KUKA KRL program: ps_b_ltb_res_c03.src, ps_b_ltb_res_c03.dat

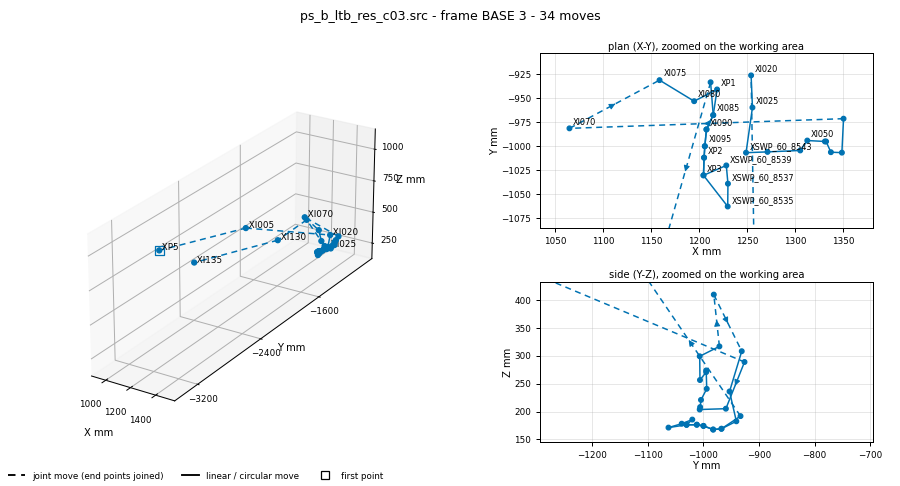
[picture p0: tool path of ps_b_ltb_res_c03.src in frame BASE 3, 34 of 34 moves have a stored position in this frame; points joined in program order, loops and branches not executed]
--- ps_b_ltb_res_c03.src ---
&ACCESS RVO1
&REL 4
&COMMENT Solda Axor LTB
&PARAM DISKPATH = KRC:\R1\Program\OLP
DEF ps_b_ltb_res_c03( )

;FOLD INI
;FOLD SPOTTECH INI
USERSPOT(#INIT)
;ENDFOLD (SPOTTECH INI)
;FOLD GRIPPERTECH INI
USER_GRP(0,DUMMY,DUMMY,GDEFAULT)
;ENDFOLD (GRIPPERTECH INI)
  ;FOLD USER INI
    ;Make your modifications here

  ;ENDFOLD (USER INI)
;ENDFOLD (INI)

; Caracterizacao dos meios de producao
; Changes: Solda Respot - AXOR - LTB
; Versao Atual: 18/02/2016
; Ferramenta: Gun C3
; Name: P13.060-R1

chk_w4_wechs_ok ( )     ; CHECK GUN C3

IF (NOT(GHOST())) THEN
IF MaxStandMenge(4) THEN
  MaxStandmengeErreicht(4)
ENDIF
IF Elektrodenwechsel(4) THEN
  e_Fraes_4 ()
ENDIF
ENDIF

;FOLD PTP P5 Vel=100 % PDAT2 Tool[4]:PINCA C3 Base[3]:Atego/Axor;%{PE}%R 8.2.20,%MKUKATPBASIS,%CMOVE,%VPTP,%P 1:PTP, 2:P5, 3:, 5:100, 7:PDAT2
$BWDSTART=FALSE
PDAT_ACT=PPDAT2
FDAT_ACT=FP5
BAS(#PTP_PARAMS,100)
PTP XP5
;ENDFOLD

;FOLD OUT 3380 'Perfil Livre Estacao' State=FALSE ;%{PE}%R 8.2.20,%MKUKATPBASIS,%COUT,%VOUTX,%P 2:3380, 3:Perfil Livre Estacao, 5:FALSE, 6:
$OUT[3380]=FALSE
;ENDFOLD

;FOLD ; Liga intertravamento 12 com R5;%{PE}%R 8.2.20,%MKUKATPBASIS,%CCOMMENT,%VNORMAL,%P 2:Liga  intertravamento  12  com  R5
;ENDFOLD
;FOLD Collision.Monitoring_12_On ;%{PE}%MKUKATPUSER
COLLSTOP( 12, 1 ) ;not Interrupt-Controlled
;ENDFOLD

;FOLD ; Liga intertravamento 13 com R5;%{PE}%R 8.2.20,%MKUKATPBASIS,%CCOMMENT,%VNORMAL,%P 2:Liga  intertravamento  13  com  R5
;ENDFOLD
;FOLD Collision.Monitoring_13_On ;%{PE}%MKUKATPUSER
COLLSTOP( 13, 1 ) ;not Interrupt-Controlled
;ENDFOLD

;FOLD PTP l005 CONT Vel=100 % P_OLP2 Tool[4]:PINCA C3 Base[3]:Atego/Axor;%{PE}%R 8.2.20,%MKUKATPBASIS,%CMOVE,%VPTP,%P 1:PTP, 2:l005, 3:C_DIS, 5:100, 7:P_OLP2
$BWDSTART=FALSE
PDAT_ACT=PP_OLP2
FDAT_ACT=Fl005
BAS(#PTP_PARAMS,100)
PTP Xl005 C_DIS
;ENDFOLD
;FOLD PTP l020 CONT Vel=100 % PDAT3 Tool[4]:PINCA C3 Base[3]:Atego/Axor;%{PE}%R 8.2.20,%MKUKATPBASIS,%CMOVE,%VPTP,%P 1:PTP, 2:l020, 3:C_DIS, 5:100, 7:PDAT3
$BWDSTART=FALSE
PDAT_ACT=PPDAT3
FDAT_ACT=Fl020
BAS(#PTP_PARAMS,100)
PTP Xl020 C_DIS
;ENDFOLD
;FOLD LIN l025 CONT Vel=2 m/s L_OLP3 Tool[4]:PINCA C3 Base[3]:Atego/Axor;%{PE}%R 8.2.20,%MKUKATPBASIS,%CMOVE,%VLIN,%P 1:LIN, 2:l025, 3:C_DIS C_DIS, 5:2, 7:L_OLP3
$BWDSTART=FALSE
LDAT_ACT=LL_OLP3
FDAT_ACT=Fl025
BAS(#CP_PARAMS,2)
LIN Xl025 C_DIS C_DIS
;ENDFOLD

;FOLD ; SWP_60_8543;%{PE}%R 4.1.16,%MKUKATPBASIS,%CCOMMENT,%VNORMAL,%P 2:SWP_60_8543
;ENDFOLD
;FOLD LIN SWP_60_8543 L_OLP4 SPOT Gun=3 RETR CLS PgNo1=196 ACTIVE=1 Tool[4]:PINCA C3 Base[3]:Atego/Axor;%{PE}%R 8.2.2,%MKUKATPSPOT,%CSPOT,%VLIN,%P 1:LIN, 2:SWP_60_8543, 3:, 5:2, 7:L_OLP4, 10:3, 12:#FIRST, 14:#CLO, 16:196, 18:1, 20:0, 22:0, 24:1, 25:NORMAL
$BWDSTART=FALSE
LDAT_ACT=LL_OLP4
FDAT_ACT=FSWP_60_8543
BAS(#CP_PARAMS,LL_OLP4.VEL)
S_ACT.GUN=3
S_ACT.PAIR=SDEFAULT.PAIR
S_ACT.RETR=#CLO
S_ACT.CLO_TM=1
S_ACT.PGNO1=196
S_ACT.PGNO2=SDEFAULT.PGNO2
S_ACT.PRESS1=SDEFAULT.PRESS1
S_ACT.PRESS2=SDEFAULT.PRESS2
S_READY=FALSE
LIN XSWP_60_8543
USERSPOT(#SPOT, S_ACT)
WAIT FOR S_READY
;ENDFOLD

;FOLD ; SWP_60_8545;%{PE}%R 4.1.16,%MKUKATPBASIS,%CCOMMENT,%VNORMAL,%P 2:SWP_60_8545
;ENDFOLD
;FOLD LIN SWP_60_8545 L_OLP8 SPOT Gun=3 RETR CLS PgNo1=196 ACTIVE=1 Tool[4]:PINCA C3 Base[3]:Atego/Axor;%{PE}%R 8.2.2,%MKUKATPSPOT,%CSPOT,%VLIN,%P 1:LIN, 2:SWP_60_8545, 3:, 5:2, 7:L_OLP8, 10:3, 12:#FIRST, 14:#CLO, 16:196, 18:1, 20:0, 22:0, 24:1, 25:NORMAL
$BWDSTART=FALSE
LDAT_ACT=LL_OLP8
FDAT_ACT=FSWP_60_8545
BAS(#CP_PARAMS,LL_OLP8.VEL)
S_ACT.GUN=3
S_ACT.PAIR=SDEFAULT.PAIR
S_ACT.RETR=#CLO
S_ACT.CLO_TM=1
S_ACT.PGNO1=196
S_ACT.PGNO2=SDEFAULT.PGNO2
S_ACT.PRESS1=SDEFAULT.PRESS1
S_ACT.PRESS2=SDEFAULT.PRESS2
S_READY=FALSE
LIN XSWP_60_8545
USERSPOT(#SPOT, S_ACT)
WAIT FOR S_READY
;ENDFOLD

;FOLD ; SWP_60_8547;%{PE}%R 4.1.16,%MKUKATPBASIS,%CCOMMENT,%VNORMAL,%P 2:SWP_60_8547
;ENDFOLD
;FOLD LIN SWP_60_8547 L_OLP9 SPOT Gun=3 RETR CLS PgNo1=196 ACTIVE=1 Tool[4]:PINCA C3 Base[3]:Atego/Axor;%{PE}%R 8.2.2,%MKUKATPSPOT,%CSPOT,%VLIN,%P 1:LIN, 2:SWP_60_8547, 3:, 5:2, 7:L_OLP9, 10:3, 12:#FIRST, 14:#CLO, 16:196, 18:1, 20:0, 22:0, 24:1, 25:NORMAL
$BWDSTART=FALSE
LDAT_ACT=LL_OLP9
FDAT_ACT=FSWP_60_8547
BAS(#CP_PARAMS,LL_OLP9.VEL)
S_ACT.GUN=3
S_ACT.PAIR=SDEFAULT.PAIR
S_ACT.RETR=#CLO
S_ACT.CLO_TM=1
S_ACT.PGNO1=196
S_ACT.PGNO2=SDEFAULT.PGNO2
S_ACT.PRESS1=SDEFAULT.PRESS1
S_ACT.PRESS2=SDEFAULT.PRESS2
S_READY=FALSE
LIN XSWP_60_8547
USERSPOT(#SPOT, S_ACT)
WAIT FOR S_READY
;ENDFOLD

;FOLD LIN l050 CONT Vel=2 m/s L_OLP10 Tool[4]:PINCA C3 Base[3]:Atego/Axor;%{PE}%R 8.2.20,%MKUKATPBASIS,%CMOVE,%VLIN,%P 1:LIN, 2:l050, 3:C_DIS C_DIS, 5:2, 7:L_OLP10
$BWDSTART=FALSE
LDAT_ACT=LL_OLP10
FDAT_ACT=Fl050
BAS(#CP_PARAMS,2)
LIN Xl050 C_DIS C_DIS
;ENDFOLD
;FOLD LIN l055 CONT Vel=2 m/s L_OLP11 Tool[4]:PINCA C3 Base[3]:Atego/Axor;%{PE}%R 8.2.20,%MKUKATPBASIS,%CMOVE,%VLIN,%P 1:LIN, 2:l055, 3:C_DIS C_DIS, 5:2, 7:L_OLP11
$BWDSTART=FALSE
LDAT_ACT=LL_OLP11
FDAT_ACT=Fl055
BAS(#CP_PARAMS,2)
LIN Xl055 C_DIS C_DIS
;ENDFOLD
;FOLD LIN l025S CONT Vel=2 m/s L_OLP12 Tool[4]:PINCA C3 Base[3]:Atego/Axor;%{PE}%R 8.2.20,%MKUKATPBASIS,%CMOVE,%VLIN,%P 1:LIN, 2:l025S, 3:C_DIS C_DIS, 5:2, 7:L_OLP12
$BWDSTART=FALSE
LDAT_ACT=LL_OLP12
FDAT_ACT=Fl025S
BAS(#CP_PARAMS,2)
LIN Xl025S C_DIS C_DIS
;ENDFOLD

;FOLD ; SWP_60_8549;%{PE}%R 4.1.16,%MKUKATPBASIS,%CCOMMENT,%VNORMAL,%P 2:SWP_60_8549
;ENDFOLD
;FOLD LIN SWP_60_8549 L_OLP13 SPOT Gun=3 RETR CLS PgNo1=196 ACTIVE=1 Tool[4]:PINCA C3 Base[3]:Atego/Axor;%{PE}%R 8.2.2,%MKUKATPSPOT,%CSPOT,%VLIN,%P 1:LIN, 2:SWP_60_8549, 3:, 5:2, 7:L_OLP13, 10:3, 12:#FIRST, 14:#CLO, 16:196, 18:1, 20:0, 22:0, 24:1, 25:NORMAL
$BWDSTART=FALSE
LDAT_ACT=LL_OLP13
FDAT_ACT=FSWP_60_8549
BAS(#CP_PARAMS,LL_OLP13.VEL)
S_ACT.GUN=3
S_ACT.PAIR=SDEFAULT.PAIR
S_ACT.RETR=#CLO
S_ACT.CLO_TM=1
S_ACT.PGNO1=196
S_ACT.PGNO2=SDEFAULT.PGNO2
S_ACT.PRESS1=SDEFAULT.PRESS1
S_ACT.PRESS2=SDEFAULT.PRESS2
S_READY=FALSE
LIN XSWP_60_8549
USERSPOT(#SPOT, S_ACT)
WAIT FOR S_READY
;ENDFOLD

;FOLD ; SWP_60_8551;%{PE}%R 4.1.16,%MKUKATPBASIS,%CCOMMENT,%VNORMAL,%P 2:SWP_60_8551
;ENDFOLD
;FOLD LIN SWP_60_8551 L_OLP14 SPOT Gun=3 RETR OPN PgNo1=196 ACTIVE=1 Tool[4]:PINCA C3 Base[3]:Atego/Axor;%{PE}%R 8.2.2,%MKUKATPSPOT,%CSPOT,%VLIN,%P 1:LIN, 2:SWP_60_8551, 3:, 5:2, 7:L_OLP14, 10:3, 12:#FIRST, 14:#OPN, 16:196, 18:1, 20:0, 22:0, 24:1, 25:NORMAL
$BWDSTART=FALSE
LDAT_ACT=LL_OLP14
FDAT_ACT=FSWP_60_8551
BAS(#CP_PARAMS,LL_OLP14.VEL)
S_ACT.GUN=3
S_ACT.PAIR=SDEFAULT.PAIR
S_ACT.RETR=#OPN
S_ACT.CLO_TM=1
S_ACT.PGNO1=196
S_ACT.PGNO2=SDEFAULT.PGNO2
S_ACT.PRESS1=SDEFAULT.PRESS1
S_ACT.PRESS2=SDEFAULT.PRESS2
S_READY=FALSE
LIN XSWP_60_8551
USERSPOT(#SPOT, S_ACT)
WAIT FOR S_READY
;ENDFOLD

;FOLD LIN l065 CONT Vel=2 m/s L_OLP15 Tool[4]:PINCA C3 Base[3]:Atego/Axor;%{PE}%R 8.2.20,%MKUKATPBASIS,%CMOVE,%VLIN,%P 1:LIN, 2:l065, 3:C_DIS C_DIS, 5:2, 7:L_OLP15
$BWDSTART=FALSE
LDAT_ACT=LL_OLP15
FDAT_ACT=Fl065
BAS(#CP_PARAMS,2)
LIN Xl065 C_DIS C_DIS
;ENDFOLD
;FOLD PTP l070 CONT Vel=100 % P_OLP5 Tool[4]:PINCA C3 Base[3]:Atego/Axor;%{PE}%R 8.2.20,%MKUKATPBASIS,%CMOVE,%VPTP,%P 1:PTP, 2:l070, 3:C_DIS, 5:100, 7:P_OLP5
$BWDSTART=FALSE
PDAT_ACT=PP_OLP5
FDAT_ACT=Fl070
BAS(#PTP_PARAMS,100)
PTP Xl070 C_DIS
;ENDFOLD
;FOLD PTP l075 CONT Vel=100 % P_OLP6 Tool[4]:PINCA C3 Base[3]:Atego/Axor;%{PE}%R 8.2.20,%MKUKATPBASIS,%CMOVE,%VPTP,%P 1:PTP, 2:l075, 3:C_DIS, 5:100, 7:P_OLP6
$BWDSTART=FALSE
PDAT_ACT=PP_OLP6
FDAT_ACT=Fl075
BAS(#PTP_PARAMS,100)
PTP Xl075 C_DIS
;ENDFOLD
;FOLD LIN l080 CONT Vel=2 m/s L_OLP16 Tool[4]:PINCA C3 Base[3]:Atego/Axor;%{PE}%R 8.2.20,%MKUKATPBASIS,%CMOVE,%VLIN,%P 1:LIN, 2:l080, 3:C_DIS C_DIS, 5:2, 7:L_OLP16
$BWDSTART=FALSE
LDAT_ACT=LL_OLP16
FDAT_ACT=Fl080
BAS(#CP_PARAMS,2)
LIN Xl080 C_DIS C_DIS
;ENDFOLD
;FOLD LIN P1 CONT Vel=2 m/s CPDAT1 Tool[4]:PINCA C3 Base[3]:Atego/Axor;%{PE}%R 8.2.20,%MKUKATPBASIS,%CMOVE,%VLIN,%P 1:LIN, 2:P1, 3:C_DIS C_DIS, 5:2, 7:CPDAT1
$BWDSTART=FALSE
LDAT_ACT=LCPDAT1
FDAT_ACT=FP1
BAS(#CP_PARAMS,2)
LIN XP1 C_DIS C_DIS
;ENDFOLD
;FOLD LIN l085 Vel=2 m/s L_OLP17 Tool[4]:PINCA C3 Base[3]:Atego/Axor;%{PE}%R 8.2.20,%MKUKATPBASIS,%CMOVE,%VLIN,%P 1:LIN, 2:l085, 3:, 5:2, 7:L_OLP17
$BWDSTART=FALSE
LDAT_ACT=LL_OLP17
FDAT_ACT=Fl085
BAS(#CP_PARAMS,2)
LIN Xl085
;ENDFOLD
;FOLD LIN l090 CONT Vel=2 m/s L_OLP18 Tool[4]:PINCA C3 Base[3]:Atego/Axor;%{PE}%R 8.2.20,%MKUKATPBASIS,%CMOVE,%VLIN,%P 1:LIN, 2:l090, 3:C_DIS C_DIS, 5:2, 7:L_OLP18
$BWDSTART=FALSE
LDAT_ACT=LL_OLP18
FDAT_ACT=Fl090
BAS(#CP_PARAMS,2)
LIN Xl090 C_DIS C_DIS
;ENDFOLD
;FOLD LIN l095 CONT Vel=2 m/s L_OLP19 Tool[4]:PINCA C3 Base[3]:Atego/Axor;%{PE}%R 8.2.20,%MKUKATPBASIS,%CMOVE,%VLIN,%P 1:LIN, 2:l095, 3:C_DIS C_DIS, 5:2, 7:L_OLP19
$BWDSTART=FALSE
LDAT_ACT=LL_OLP19
FDAT_ACT=Fl095
BAS(#CP_PARAMS,2)
LIN Xl095 C_DIS C_DIS
;ENDFOLD
;FOLD LIN P2 CONT Vel=2 m/s CPDAT2 Tool[4]:PINCA C3 Base[3]:Atego/Axor;%{PE}%R 8.2.20,%MKUKATPBASIS,%CMOVE,%VLIN,%P 1:LIN, 2:P2, 3:C_DIS C_DIS, 5:2, 7:CPDAT2
$BWDSTART=FALSE
LDAT_ACT=LCPDAT2
FDAT_ACT=FP2
BAS(#CP_PARAMS,2)
LIN XP2 C_DIS C_DIS
;ENDFOLD
;FOLD LIN P3 CONT Vel=2 m/s CPDAT3 Tool[4]:PINCA C3 Base[3]:Atego/Axor;%{PE}%R 8.2.20,%MKUKATPBASIS,%CMOVE,%VLIN,%P 1:LIN, 2:P3, 3:C_DIS C_DIS, 5:2, 7:CPDAT3
$BWDSTART=FALSE
LDAT_ACT=LCPDAT3
FDAT_ACT=FP3
BAS(#CP_PARAMS,2)
LIN XP3 C_DIS C_DIS
;ENDFOLD

;FOLD ; SWP_60_8535;%{PE}%R 8.2.20,%MKUKATPBASIS,%CCOMMENT,%VNORMAL,%P 2:SWP_60_8535
;ENDFOLD
;FOLD LIN SWP_60_8535 L_OLP30 SPOT Gun=3 RETR CLS PgNo1=197 ACTIVE=1 Tool[4]:PINCA C3 Base[3]:Atego/Axor;%{PE}%R 8.2.2,%MKUKATPSPOT,%CSPOT,%VLIN,%P 1:LIN, 2:SWP_60_8535, 3:, 5:2, 7:L_OLP30, 10:3, 12:#FIRST, 14:#CLO, 16:197, 18:1, 20:0, 22:0, 24:1, 25:NORMAL
$BWDSTART=FALSE
LDAT_ACT=LL_OLP30
FDAT_ACT=FSWP_60_8535
BAS(#CP_PARAMS,LL_OLP30.VEL)
S_ACT.GUN=3
S_ACT.PAIR=SDEFAULT.PAIR
S_ACT.RETR=#CLO
S_ACT.CLO_TM=1
S_ACT.PGNO1=197
S_ACT.PGNO2=SDEFAULT.PGNO2
S_ACT.PRESS1=SDEFAULT.PRESS1
S_ACT.PRESS2=SDEFAULT.PRESS2
S_READY=FALSE
LIN XSWP_60_8535
USERSPOT(#SPOT, S_ACT)
WAIT FOR S_READY
;ENDFOLD

;FOLD ; SWP_60_8537;%{PE}%R 8.2.20,%MKUKATPBASIS,%CCOMMENT,%VNORMAL,%P 2:SWP_60_8537
;ENDFOLD
;FOLD LIN SWP_60_8537 L_OLP31 SPOT Gun=3 RETR CLS PgNo1=197 ACTIVE=1 Tool[4]:PINCA C3 Base[3]:Atego/Axor;%{PE}%R 8.2.2,%MKUKATPSPOT,%CSPOT,%VLIN,%P 1:LIN, 2:SWP_60_8537, 3:, 5:2, 7:L_OLP31, 10:3, 12:#FIRST, 14:#CLO, 16:197, 18:1, 20:0, 22:0, 24:1, 25:NORMAL
$BWDSTART=FALSE
LDAT_ACT=LL_OLP31
FDAT_ACT=FSWP_60_8537
BAS(#CP_PARAMS,LL_OLP31.VEL)
S_ACT.GUN=3
S_ACT.PAIR=SDEFAULT.PAIR
S_ACT.RETR=#CLO
S_ACT.CLO_TM=1
S_ACT.PGNO1=197
S_ACT.PGNO2=SDEFAULT.PGNO2
S_ACT.PRESS1=SDEFAULT.PRESS1
S_ACT.PRESS2=SDEFAULT.PRESS2
S_READY=FALSE
LIN XSWP_60_8537
USERSPOT(#SPOT, S_ACT)
WAIT FOR S_READY
;ENDFOLD

;FOLD ; SWP_60_8539;%{PE}%R 4.1.16,%MKUKATPBASIS,%CCOMMENT,%VNORMAL,%P 2:SWP_60_8539
;ENDFOLD
;FOLD LIN SWP_60_8539 L_OLP20 SPOT Gun=3 RETR OPN PgNo1=197 ACTIVE=1 Tool[4]:PINCA C3 Base[3]:Atego/Axor;%{PE}%R 8.2.2,%MKUKATPSPOT,%CSPOT,%VLIN,%P 1:LIN, 2:SWP_60_8539, 3:, 5:2, 7:L_OLP20, 10:3, 12:#FIRST, 14:#OPN, 16:197, 18:1, 20:0, 22:0, 24:1, 25:NORMAL
$BWDSTART=FALSE
LDAT_ACT=LL_OLP20
FDAT_ACT=FSWP_60_8539
BAS(#CP_PARAMS,LL_OLP20.VEL)
S_ACT.GUN=3
S_ACT.PAIR=SDEFAULT.PAIR
S_ACT.RETR=#OPN
S_ACT.CLO_TM=1
S_ACT.PGNO1=197
S_ACT.PGNO2=SDEFAULT.PGNO2
S_ACT.PRESS1=SDEFAULT.PRESS1
S_ACT.PRESS2=SDEFAULT.PRESS2
S_READY=FALSE
LIN XSWP_60_8539
USERSPOT(#SPOT, S_ACT)
WAIT FOR S_READY
;ENDFOLD

;FOLD LIN P4 CONT Vel=2 m/s CPDAT4 Tool[4]:PINCA C3 Base[3]:Atego/Axor;%{PE}%R 8.2.20,%MKUKATPBASIS,%CMOVE,%VLIN,%P 1:LIN, 2:P4, 3:C_DIS C_DIS, 5:2, 7:CPDAT4
$BWDSTART=FALSE
LDAT_ACT=LCPDAT4
FDAT_ACT=FP4
BAS(#CP_PARAMS,2)
LIN XP4 C_DIS C_DIS
;ENDFOLD
;FOLD LIN l100 CONT Vel=2 m/s L_OLP23 Tool[4]:PINCA C3 Base[3]:Atego/Axor;%{PE}%R 8.2.20,%MKUKATPBASIS,%CMOVE,%VLIN,%P 1:LIN, 2:l100, 3:C_DIS C_DIS, 5:2, 7:L_OLP23
$BWDSTART=FALSE
LDAT_ACT=LL_OLP23
FDAT_ACT=Fl100
BAS(#CP_PARAMS,2)
LIN Xl100 C_DIS C_DIS
;ENDFOLD
;FOLD LIN l105 CONT Vel=2 m/s L_OLP24 Tool[4]:PINCA C3 Base[3]:Atego/Axor;%{PE}%R 8.2.20,%MKUKATPBASIS,%CMOVE,%VLIN,%P 1:LIN, 2:l105, 3:C_DIS C_DIS, 5:2, 7:L_OLP24
$BWDSTART=FALSE
LDAT_ACT=LL_OLP24
FDAT_ACT=Fl105
BAS(#CP_PARAMS,2)
LIN Xl105 C_DIS C_DIS
;ENDFOLD
;FOLD LIN l110 CONT Vel=2 m/s L_OLP25 Tool[4]:PINCA C3 Base[3]:Atego/Axor;%{PE}%R 8.2.20,%MKUKATPBASIS,%CMOVE,%VLIN,%P 1:LIN, 2:l110, 3:C_DIS C_DIS, 5:2, 7:L_OLP25
$BWDSTART=FALSE
LDAT_ACT=LL_OLP25
FDAT_ACT=Fl110
BAS(#CP_PARAMS,2)
LIN Xl110 C_DIS C_DIS
;ENDFOLD
;FOLD LIN l115  Vel=2.00 m/s L_OLP26 Tool[4]:Gun C03 Base[3]:Atego/Axor;%{PE}%R8.2.19,%MKUKATPBASIS,%CMOVE,%VLIN,%P 1:LIN, 2:l115, 3: , 5:2.00, 7:L_OLP26
$BWDSTART = FALSE
LDAT_ACT= LL_OLP26
FDAT_ACT= Fl115
BAS(#CP_PARAMS,2.00)
LIN Xl115
;ENDFOLD
;FOLD LIN l120 CONT Vel=2 m/s L_OLP27 Tool[4]:PINCA C3 Base[3]:Atego/Axor;%{PE}%R 8.2.20,%MKUKATPBASIS,%CMOVE,%VLIN,%P 1:LIN, 2:l120, 3:C_DIS C_DIS, 5:2, 7:L_OLP27
$BWDSTART=FALSE
LDAT_ACT=LL_OLP27
FDAT_ACT=Fl120
BAS(#CP_PARAMS,2)
LIN Xl120 C_DIS C_DIS
;ENDFOLD
;FOLD PTP l125 CONT Vel=100 % PDAT4 Tool[4]:PINCA C3 Base[3]:Atego/Axor;%{PE}%R 8.2.20,%MKUKATPBASIS,%CMOVE,%VPTP,%P 1:PTP, 2:l125, 3:C_DIS, 5:100, 7:PDAT4
$BWDSTART=FALSE
PDAT_ACT=PPDAT4
FDAT_ACT=Fl125
BAS(#PTP_PARAMS,100)
PTP Xl125 C_DIS
;ENDFOLD
;FOLD PTP l130 CONT Vel=100 % PDAT5 Tool[4]:PINCA C3 Base[3]:Atego/Axor;%{PE}%R 8.2.20,%MKUKATPBASIS,%CMOVE,%VPTP,%P 1:PTP, 2:l130, 3:C_DIS, 5:100, 7:PDAT5
$BWDSTART=FALSE
PDAT_ACT=PPDAT5
FDAT_ACT=Fl130
BAS(#PTP_PARAMS,100)
PTP Xl130 C_DIS
;ENDFOLD
;FOLD PTP l135 Vel=100 % P_OLP7 Tool[4]:PINCA C3 Base[3]:Atego/Axor;%{PE}%R 8.2.20,%MKUKATPBASIS,%CMOVE,%VPTP,%P 1:PTP, 2:l135, 3:, 5:100, 7:P_OLP7
$BWDSTART=FALSE
PDAT_ACT=PP_OLP7
FDAT_ACT=Fl135
BAS(#PTP_PARAMS,100)
PTP Xl135
;ENDFOLD

;FOLD ; Desliga intertravamento 12 com R5;%{PE}%R 8.2.20,%MKUKATPBASIS,%CCOMMENT,%VNORMAL,%P 2:Desliga  intertravamento  12  com  R5
;ENDFOLD
;FOLD Collision.Monitoring_12_Off . ;%{PE}%MKUKATPUSER
COLLSTOP( 12, 2+0 )
;ENDFOLD

;FOLD ; Desliga intertravamento 13 com R5;%{PE}%R 8.2.20,%MKUKATPBASIS,%CCOMMENT,%VNORMAL,%P 2:Desliga  intertravamento  13  com  R5
;ENDFOLD
;FOLD Collision.Monitoring_13_Off . ;%{PE}%MKUKATPUSER
COLLSTOP( 13, 2+0 )
;ENDFOLD

end_weld_respot ()

IF (NOT(GHOST())) THEN
IF FraesAnf(4) THEN
  f_Fraes_4 ()
ENDIF
ENDIF

END

--- ps_b_ltb_res_c03.dat ---
&ACCESS RVO1
&REL 4
&COMMENT Solda Axor LTB
&PARAM DISKPATH = KRC:\R1\Program\OLP
DEFDAT ps_b_ltb_res_c03
;FOLD EXTERNAL DECLARATIONS;%{PE}%MKUKATPBASIS,%CEXT,%VCOMMON,%P
;FOLD GRIPPERTECH EXT
EXT  H50 (INT  :IN,INT  :IN,INT  :IN,GRP_TYP  :IN )
;ENDFOLD (GRIPPERTECH EXT)
;FOLD SPOTTECH EXT
EXT  USERSPOT (S_COMMAND  :IN,SPOT_TYPE  :IN )
;ENDFOLD (SPOTTECH EXT)
;FOLD BASISTECH EXT;%{PE}%MKUKATPBASIS,%CEXT,%VEXT,%P
EXT  BAS (BAS_COMMAND  :IN,REAL  :IN )
DECL INT SUCCESS
;ENDFOLD (BASISTECH EXT)
;FOLD USER EXT;%{E}%MKUKATPUSER,%CEXT,%VEXT,%P
;Make your modifications here

;ENDFOLD (USER EXT)
;ENDFOLD (EXTERNAL DECLARATIONS)
DECL FDAT Fl005={TOOL_NO 4,BASE_NO 3,IPO_FRAME #BASE,POINT2[] " "}
DECL PDAT PP_OLP2={VEL 100.0,ACC 100.0,APO_DIST 200.0,APO_MODE #CDIS}
DECL E6POS Xl005={X 1274.78198,Y -2152.4519,Z 802.703003,A 0.067400001,B 28.0000992,C 90.0,S 2,T 11}
DECL FDAT Fl020={TOOL_NO 4,BASE_NO 3,IPO_FRAME #BASE,POINT2[] " "}
DECL E6POS Xl020={X 1253.90295,Y -926.031982,Z 289.157806,A 0.0670686066,B 27.9958591,C 89.9981689,S 18,T 11,E1 0.0,E2 0.0,E3 0.0,E4 0.0,E5 0.0,E6 0.0}
DECL FDAT Fl025={TOOL_NO 4,BASE_NO 3,IPO_FRAME #BASE,POINT2[] " "}
DECL E6POS Xl025={X 1255.30298,Y -959.498718,Z 205.282593,A 0.0679476634,B 27.99827,C 89.999649,S 18,T 11,E1 0.0,E2 0.0,E3 0.0,E4 0.0,E5 0.0,E6 0.0}
DECL LDAT LL_OLP3={VEL 2.0,ACC 100.0,APO_DIST 10.0,APO_FAC 0.0,ORI_TYP #VAR,CIRC_TYP #BASE,JERK_FAC 50.0}
DECL FDAT FSWP_60_8543={TOOL_NO 4,BASE_NO 3,IPO_FRAME #BASE,POINT2[] " "}
DECL E6POS XSWP_60_8543={X 1248.61499,Y -1006.54199,Z 203.796402,A -0.129490495,B 27.9995594,C 92.4205933,S 18,T 11,E1 0.0,E2 0.0,E3 0.0,E4 0.0,E5 0.0,E6 0.0}
DECL LDAT LL_OLP4={VEL 2.0,ACC 100.0,APO_DIST 0.0,APO_FAC 0.0,ORI_TYP #VAR,CIRC_TYP #BASE,JERK_FAC 50.0}
DECL FDAT FSWP_60_8545={TOOL_NO 4,BASE_NO 3,IPO_FRAME #BASE,POINT2[] " "}
DECL E6POS XSWP_60_8545={X 1270.98096,Y -1005.711,Z 208.158401,A -0.129547194,B 27.9999104,C 92.419487,S 18,T 11,E1 0.0,E2 0.0,E3 0.0,E4 0.0,E5 0.0,E6 0.0}
DECL LDAT LL_OLP8={VEL 2.0,ACC 100.0,APO_DIST 0.0,APO_FAC 0.0,ORI_TYP #VAR,CIRC_TYP #BASE,JERK_FAC 50.0}
DECL FDAT FSWP_60_8547={TOOL_NO 4,BASE_NO 3,IPO_FRAME #BASE,POINT2[] " "}
DECL E6POS XSWP_60_8547={X 1305.07202,Y -1004.21399,Z 221.033096,A 0.224301994,B 35.0479698,C 92.027832,S 18,T 11,E1 0.0,E2 0.0,E3 0.0,E4 0.0,E5 0.0,E6 0.0}
DECL LDAT LL_OLP9={VEL 2.0,ACC 100.0,APO_DIST 0.0,APO_FAC 0.0,ORI_TYP #VAR,CIRC_TYP #BASE,JERK_FAC 50.0}
DECL FDAT Fl050={TOOL_NO 4,BASE_NO 3,IPO_FRAME #BASE,POINT2[] " "}
DECL E6POS Xl050={X 1312.42297,Y -993.888977,Z 240.986099,A 0.0672914535,B 27.9993992,C 90.0008469,S 18,T 11,E1 0.0,E2 0.0,E3 0.0,E4 0.0,E5 0.0,E6 0.0}
DECL LDAT LL_OLP10={VEL 2.0,ACC 100.0,APO_DIST 5.0,APO_FAC 0.0,ORI_TYP #VAR,CIRC_TYP #BASE,JERK_FAC 50.0}
DECL FDAT Fl055={TOOL_NO 4,BASE_NO 3,IPO_FRAME #BASE,POINT2[] " "}
DECL E6POS Xl055={X 1330.77405,Y -994.846619,Z 273.997803,A 0.0951634571,B 19.9996204,C 90.0010986,S 18,T 11,E1 0.0,E2 0.0,E3 0.0,E4 0.0,E5 0.0,E6 0.0}
DECL LDAT LL_OLP11={VEL 2.0,ACC 100.0,APO_DIST 5.0,APO_FAC 0.0,ORI_TYP #VAR,CIRC_TYP #BASE,JERK_FAC 50.0}
DECL FDAT Fl025S={TOOL_NO 4,BASE_NO 3,IPO_FRAME #BASE,POINT2[] " "}
DECL E6POS Xl025S={X 1331.99402,Y -994.88147,Z 271.029297,A 0.0962694436,B -0.00231891288,C 89.9995804,S 18,T 11,E1 0.0,E2 0.0,E3 0.0,E4 0.0,E5 0.0,E6 0.0}
DECL LDAT LL_OLP12={VEL 2.0,ACC 100.0,APO_DIST 5.0,APO_FAC 0.0,ORI_TYP #VAR,CIRC_TYP #BASE,JERK_FAC 50.0}
DECL FDAT FSWP_60_8549={TOOL_NO 4,BASE_NO 3,IPO_FRAME #BASE,POINT2[] " "}
DECL E6POS XSWP_60_8549={X 1336.99695,Y -1006.02899,Z 256.759003,A 2.13942194,B -0.046111729,C 91.2335129,S 18,T 3,E1 0.0,E2 0.0,E3 0.0,E4 0.0,E5 0.0,E6 0.0}
DECL LDAT LL_OLP13={VEL 2.0,ACC 100.0,APO_DIST 0.0,APO_FAC 0.0,ORI_TYP #VAR,CIRC_TYP #BASE,JERK_FAC 50.0}
DECL FDAT FSWP_60_8551={TOOL_NO 4,BASE_NO 3,IPO_FRAME #BASE,POINT2[] " "}
DECL E6POS XSWP_60_8551={X 1348.448,Y -1006.50098,Z 299.4151,A 0.931857288,B -0.001559027,C 90.0008163,S 18,T 11,E1 0.0,E2 0.0,E3 0.0,E4 0.0,E5 0.0,E6 0.0}
DECL LDAT LL_OLP14={VEL 2.0,ACC 100.0,APO_DIST 0.0,APO_FAC 0.0,ORI_TYP #VAR,CIRC_TYP #BASE,JERK_FAC 50.0}
DECL FDAT Fl065={TOOL_NO 4,BASE_NO 3,IPO_FRAME #BASE,POINT2[] " "}
DECL E6POS Xl065={X 1350.17297,Y -971.119019,Z 317.191986,A 0.107299998,B 0.0,C 90.0,S 2,T 3}
DECL LDAT LL_OLP15={VEL 2.0,ACC 100.0,APO_DIST 10.0,APO_FAC 0.0,ORI_TYP #VAR,CIRC_TYP #BASE,JERK_FAC 50.0}
DECL FDAT Fl070={TOOL_NO 4,BASE_NO 3,IPO_FRAME #BASE,POINT2[] " "}
DECL PDAT PP_OLP5={VEL 100.0,ACC 100.0,APO_DIST 30.0,APO_MODE #CDIS}
DECL E6POS Xl070={X 1064.72302,Y -981.197998,Z 410.233002,A 0.067400001,B 28.0,C 90.0,S 2,T 11}
DECL FDAT Fl075={TOOL_NO 4,BASE_NO 3,IPO_FRAME #BASE,POINT2[] " "}
DECL PDAT PP_OLP6={VEL 100.0,ACC 100.0,APO_DIST 10.0,APO_MODE #CDIS}
DECL E6POS Xl075={X 1158.53699,Y -930.995972,Z 308.523712,A -79.3087234,B 43.2878685,C 15.4422798,S 18,T 11,E1 0.0,E2 0.0,E3 0.0,E4 0.0,E5 0.0,E6 0.0}
DECL FDAT Fl080={TOOL_NO 4,BASE_NO 3,IPO_FRAME #BASE,POINT2[] " "}
DECL E6POS Xl080={X 1194.58398,Y -952.924805,Z 236.176804,A -83.9426422,B 34.0680809,C 12.1901903,S 18,T 11,E1 0.0,E2 0.0,E3 0.0,E4 0.0,E5 0.0,E6 0.0}
DECL LDAT LL_OLP16={VEL 2.0,ACC 90.0,APO_DIST 5.0,APO_FAC 0.0,ORI_TYP #VAR,CIRC_TYP #BASE,JERK_FAC 50.0}
DECL FDAT Fl085={TOOL_NO 4,BASE_NO 3,IPO_FRAME #BASE,POINT2[] " "}
DECL E6POS Xl085={X 1214.45496,Y -967.418823,Z 169.231796,A -85.3647232,B 33.5413094,C 11.77003,S 18,T 11,E1 0.0,E2 0.0,E3 0.0,E4 0.0,E5 0.0,E6 0.0}
DECL LDAT LL_OLP17={VEL 2.0,ACC 90.0,APO_DIST 0.0,APO_FAC 0.0,ORI_TYP #VAR,CIRC_TYP #BASE,JERK_FAC 50.0}
DECL FDAT Fl090={TOOL_NO 4,BASE_NO 3,IPO_FRAME #BASE,POINT2[] " "}
DECL E6POS Xl090={X 1207.41296,Y -982.324219,Z 167.815506,A -86.5582275,B 28.5024891,C 11.1536798,S 18,T 11,E1 0.0,E2 0.0,E3 0.0,E4 0.0,E5 0.0,E6 0.0}
DECL LDAT LL_OLP18={VEL 2.0,ACC 90.0,APO_DIST 0.0,APO_FAC 0.0,ORI_TYP #VAR,CIRC_TYP #BASE,JERK_FAC 50.0}
DECL FDAT Fl095={TOOL_NO 4,BASE_NO 3,IPO_FRAME #BASE,POINT2[] " "}
DECL E6POS Xl095={X 1205.70496,Y -999.781921,Z 174.400696,A -88.0589981,B 22.1710796,C 10.5196896,S 18,T 11,E1 0.0,E2 0.0,E3 0.0,E4 0.0,E5 0.0,E6 0.0}
DECL LDAT LL_OLP19={VEL 2.0,ACC 90.0,APO_DIST 0.0,APO_FAC 0.0,ORI_TYP #VAR,CIRC_TYP #BASE,JERK_FAC 50.0}
DECL FDAT FSWP_60_8539={TOOL_NO 4,BASE_NO 3,IPO_FRAME #BASE,POINT2[] " "}
DECL E6POS XSWP_60_8539={X 1228.07397,Y -1019.80701,Z 185.733307,A -86.5685272,B 17.1511192,C 10.9525404,S 18,T 11,E1 0.0,E2 0.0,E3 0.0,E4 0.0,E5 0.0,E6 0.0}
DECL LDAT LL_OLP20={VEL 2.0,ACC 100.0,APO_DIST 0.0,APO_FAC 0.0,ORI_TYP #VAR,CIRC_TYP #BASE,JERK_FAC 50.0}
DECL FDAT FSWP_60_8537={TOOL_NO 4,BASE_NO 3,IPO_FRAME #BASE,POINT2[] " "}
DECL E6POS XSWP_60_8537={X 1229.78503,Y -1038.82397,Z 178.347,A -85.155838,B 16.9215202,C 11.3460102,S 18,T 11,E1 0.0,E2 0.0,E3 0.0,E4 0.0,E5 0.0,E6 0.0}
DECL FDAT FSWP_60_8535={TOOL_NO 4,BASE_NO 3,IPO_FRAME #BASE,POINT2[] " "}
DECL E6POS XSWP_60_8535={X 1229.53296,Y -1062.57898,Z 171.323593,A -85.0608063,B 16.9015503,C 11.3733501,S 18,T 11,E1 0.0,E2 0.0,E3 0.0,E4 0.0,E5 0.0,E6 0.0}
DECL FDAT Fl100={TOOL_NO 4,BASE_NO 3,IPO_FRAME #BASE,POINT2[] " "}
DECL E6POS Xl100={X 1204.92896,Y -1011.70398,Z 176.505096,A -88.2505264,B 21.2112293,C 10.44874,S 18,T 11,E1 0.0,E2 0.0,E3 0.0,E4 0.0,E5 0.0,E6 0.0}
DECL LDAT LL_OLP23={VEL 2.0,ACC 90.0,APO_DIST 0.0,APO_FAC 0.0,ORI_TYP #VAR,CIRC_TYP #BASE,JERK_FAC 50.0}
DECL FDAT Fl105={TOOL_NO 4,BASE_NO 3,IPO_FRAME #BASE,POINT2[] " "}
DECL E6POS Xl105={X 1205.70703,Y -999.784119,Z 174.397995,A -88.2506332,B 21.2111702,C 10.4488602,S 18,T 11,E1 0.0,E2 0.0,E3 0.0,E4 0.0,E5 0.0,E6 0.0}
DECL LDAT LL_OLP24={VEL 2.0,ACC 90.0,APO_DIST 0.0,APO_FAC 0.0,ORI_TYP #VAR,CIRC_TYP #BASE,JERK_FAC 50.0}
DECL FDAT Fl110={TOOL_NO 4,BASE_NO 3,IPO_FRAME #BASE,POINT2[] " "}
DECL E6POS Xl110={X 1207.41797,Y -982.322876,Z 167.813293,A -86.5583267,B 28.50243,C 11.15378,S 18,T 11,E1 0.0,E2 0.0,E3 0.0,E4 0.0,E5 0.0,E6 0.0}
DECL LDAT LL_OLP25={VEL 2.0,ACC 90.0,APO_DIST 0.0,APO_FAC 0.0,ORI_TYP #VAR,CIRC_TYP #BASE,JERK_FAC 50.0}
DECL FDAT Fl115={TOOL_NO 4,BASE_NO 3,IPO_FRAME #BASE,POINT2[] " "}
DECL E6POS Xl115={X 1214.45996,Y -967.417603,Z 169.229706,A -85.36483,B 33.5412483,C 11.7701101,S 18,T 11,E1 0.0,E2 0.0,E3 0.0,E4 0.0,E5 0.0,E6 0.0}
DECL LDAT LL_OLP26={VEL 2.0,ACC 90.0,APO_DIST 0.0,APO_FAC 0.0,ORI_TYP #VAR,CIRC_TYP #BASE,JERK_FAC 50.0}
DECL FDAT Fl120={TOOL_NO 4,BASE_NO 3,IPO_FRAME #BASE,POINT2[] " "}
DECL E6POS Xl120={X 1211.70801,Y -933.204285,Z 191.964798,A -85.3650818,B 33.5403404,C 11.7698402,S 18,T 11,E1 0.0,E2 0.0,E3 0.0,E4 0.0,E5 0.0,E6 0.0}
DECL LDAT LL_OLP27={VEL 2.0,ACC 90.0,APO_DIST 0.0,APO_FAC 0.0,ORI_TYP #VAR,CIRC_TYP #BASE,JERK_FAC 50.0}
DECL FDAT Fl125={TOOL_NO 4,BASE_NO 3,IPO_FRAME #BASE,POINT2[] " "}
DECL E6POS Xl125={X 1159.677,Y -1115.85803,Z 460.207886,A -85.3720932,B 33.5464401,C 11.7702303,S 18,T 11,E1 0.0,E2 0.0,E3 0.0,E4 0.0,E5 0.0,E6 0.0}
DECL FDAT Fl130={TOOL_NO 4,BASE_NO 3,IPO_FRAME #BASE,POINT2[] " "}
DECL E6POS Xl130={X 1184.69495,Y -1570.10803,Z 471.626404,A -84.223793,B 38.9344902,C 11.9292898,S 18,T 11,E1 0.0,E2 0.0,E3 0.0,E4 0.0,E5 0.0,E6 0.0}
DECL FDAT Fl135={TOOL_NO 4,BASE_NO 3,IPO_FRAME #BASE,POINT2[] " "}
DECL PDAT PP_OLP7={VEL 100.0,ACC 100.0,APO_DIST 30.0,APO_MODE #CDIS}
DECL E6POS Xl135={X 1198.995,Y -2692.78394,Z 729.96698,A 79.1359329,B 3.19893003,C 113.345901,S 18,T 11,E1 0.0,E2 0.0,E3 0.0,E4 0.0,E5 0.0,E6 0.0}
DECL BASIS_SUGG_T LAST_BASIS={POINT1[] "P0                      ",POINT2[] "P0                      ",CP_PARAMS[] "CPDAT0                  ",PTP_PARAMS[] "PDAT0                   ",CONT[] "                        ",CP_VEL[] "2.0                     ",PTP_VEL[] " 100                    ",SYNC_PARAMS[] "SYNCDAT                 ",SPL_NAME[] "S0                      "}
DECL E6POS XP1={X 1218.46301,Y -940.685425,Z 182.637405,A -83.6815186,B 38.8470497,C 13.7355204,S 18,T 11,E1 0.0,E2 0.0,E3 0.0,E4 0.0,E5 0.0,E6 0.0}
DECL FDAT FP1={TOOL_NO 4,BASE_NO 3,IPO_FRAME #BASE,POINT2[] " ",TQ_STATE FALSE}
DECL LDAT LCPDAT1={VEL 2.0,ACC 90.0,APO_DIST 100.0,APO_FAC 50.0,AXIS_VEL 100.0,AXIS_ACC 100.0,ORI_TYP #VAR,CIRC_TYP #BASE,JERK_FAC 50.0,GEAR_JERK 50.0,EXAX_IGN 0}
DECL E6POS XP2={X 1204.92395,Y -1011.70502,Z 176.507294,A -88.2504272,B 21.2112808,C 10.4486103,S 18,T 11,E1 0.0,E2 0.0,E3 0.0,E4 0.0,E5 0.0,E6 0.0}
DECL FDAT FP2={TOOL_NO 4,BASE_NO 3,IPO_FRAME #BASE,POINT2[] " ",TQ_STATE FALSE}
DECL LDAT LCPDAT2={VEL 2.0,ACC 90.0,APO_DIST 100.0,APO_FAC 50.0,AXIS_VEL 100.0,AXIS_ACC 100.0,ORI_TYP #VAR,CIRC_TYP #BASE,JERK_FAC 50.0,GEAR_JERK 50.0,EXAX_IGN 0}
DECL E6POS XP3={X 1204.31006,Y -1030.13,Z 176.307098,A -88.9489899,B 17.6018906,C 10.2152901,S 18,T 11,E1 0.0,E2 0.0,E3 0.0,E4 0.0,E5 0.0,E6 0.0}
DECL FDAT FP3={TOOL_NO 4,BASE_NO 3,IPO_FRAME #BASE,POINT2[] " ",TQ_STATE FALSE}
DECL LDAT LCPDAT3={VEL 2.0,ACC 90.0,APO_DIST 100.0,APO_FAC 50.0,AXIS_VEL 100.0,AXIS_ACC 100.0,ORI_TYP #VAR,CIRC_TYP #BASE,JERK_FAC 50.0,GEAR_JERK 50.0,EXAX_IGN 0}
DECL LDAT LL_OLP30={VEL 2.0,ACC 100.0,APO_DIST 0.0,APO_FAC 0.0,ORI_TYP #VAR,CIRC_TYP #BASE,JERK_FAC 50.0}
DECL LDAT LL_OLP31={VEL 2.0,ACC 100.0,APO_DIST 0.0,APO_FAC 0.0,ORI_TYP #VAR,CIRC_TYP #BASE,JERK_FAC 50.0}
DECL E6POS XP4={X 1204.31702,Y -1030.12805,Z 176.301804,A -88.9490738,B 17.60186,C 10.2155399,S 18,T 11,E1 0.0,E2 0.0,E3 0.0,E4 0.0,E5 0.0,E6 0.0}
DECL FDAT FP4={TOOL_NO 4,BASE_NO 3,IPO_FRAME #BASE,POINT2[] " ",TQ_STATE FALSE}
DECL LDAT LCPDAT4={VEL 2.0,ACC 90.0,APO_DIST 100.0,APO_FAC 50.0,AXIS_VEL 100.0,AXIS_ACC 100.0,ORI_TYP #VAR,CIRC_TYP #BASE,JERK_FAC 50.0,GEAR_JERK 50.0,EXAX_IGN 0}
DECL E6POS XP5={X 1369.85901,Y -3360.61499,Z 1113.32104,A 125.899696,B -60.7102013,C 126.314598,S 18,T 3,E1 0.0,E2 0.0,E3 0.0,E4 0.0,E5 0.0,E6 0.0}
DECL FDAT FP5={TOOL_NO 4,BASE_NO 3,IPO_FRAME #BASE,POINT2[] " ",TQ_STATE FALSE}
DECL PDAT PPDAT2={VEL 100.0,ACC 100.0,APO_DIST 100.0,APO_MODE #CDIS,GEAR_JERK 50.0}
DECL PDAT PPDAT3={VEL 100.0,ACC 100.0,APO_DIST 30.0,APO_MODE #CDIS,GEAR_JERK 50.0}
DECL SPOT_SUGG_T LAST_SPOT={GUN[] "1                       ",RETR_CMD[] "#OPN                    ",CHOISE[] "#FIRST                  ",CLO_TM[] "0                       ",PGNO1[] "1                       ",PRESS1[] "0                       ",PGNO2[] "1                       ",PRESS2[] "0                       ",SPOT_PARAMS[] "NORMAL                  "}
DECL PDAT PPDAT4={VEL 100.0,ACC 100.0,APO_DIST 10.0,APO_MODE #CDIS,GEAR_JERK 50.0}
DECL PDAT PPDAT5={VEL 100.0,ACC 100.0,APO_DIST 30.0,APO_MODE #CDIS,GEAR_JERK 50.0}
ENDDAT
